(*

.. <legal notes>

legal notes
=================
| SPDX-FileCopyrightText: © 2026 Oleksandr Tiutyk <trofimich@gmail.com>
| SPDX-License-Identifier: LGPL-3.0-only
| For details check: LGPL-3.0-only_

.. _LGPL-3.0-only: https://www.gnu.org/licenses/lgpl-3.0.en.html

.. </legal notes>

*)

INTERFACE ISimpleDevice EXTENDS IDevice

END_INTERFACE

(* stored: Version 1.1.0.1
   Itf ISimpleDevice: Id {15135d0b-b078-4046-91ab-232b065f7af4} *)
